FUNCTION_BLOCK CoEResetTask IMPLEMENTS I_Task, I_Cyclic, I_Object, I_Abortable, I_Abortable, I_Resettable
VAR
	mcReset : Tc2_MC2.MC_Reset;
	_Axis : REFERENCE TO Tc2_MC2.AXIS_REF;
END_VAR

{analysis -2}

METHOD Abort : HRESULT
mcReset.Execute := FALSE;
END_METHOD

PROPERTY AxisRef : reference to Axis_Ref
GET // PUBLIC
AxisRef REF= _Axis;
END_GET
SET
_Axis REF= AxisRef;
END_SET
END_PROPERTY

PROPERTY Busy : BOOL
GET
Busy := mcReset.Busy;
END_GET
END_PROPERTY

METHOD Cycle : HRESULT
VAR_INPUT
END_VAR
mcReset(Axis := _Axis);
mcReset.Execute := FALSE;
END_METHOD

PROPERTY Done : BOOL
GET
Done := mcReset.Done;
END_GET
END_PROPERTY

PROPERTY Error : BOOL
GET
Error := mcReset.Error;
END_GET
END_PROPERTY

METHOD RegisterWithParent
VAR_INPUT
	Parent	: I_HostObjects;
END_VAR
Parent.RegisterAbortable(THIS^);
Parent.RegisterCyclic(THIS^);
Parent.RegisterTask(THIS^);
Parent.RegisterResettable(THIS^);
END_METHOD

METHOD Reset : HRESULT
VAR_INPUT
END_VAR
IF mcReset.Execute THEN
	Reset := -1;
ELSE
	mcReset.Execute := TRUE;
END_IF
END_METHOD

END_FUNCTION_BLOCK

(* stored: Version 1.1.0.1
   POU CoEResetTask: Id {ea00788b-a7e2-4ddb-a987-8527d11bfcf5}, SpecialFunc None
   Method Abort: Id {175585a1-cdb8-4dd4-9630-03b10e9f2656}
   Property AxisRef: Id {b3b662e8-3ce3-48c8-a8d0-fc2d4bd302cd}
   Get Get: Id {23224859-c01c-495b-a166-81f774c86dc0}
   Set Set: Id {378228be-d0bf-44b9-a6ef-d5a5e53194bf}
   Property Busy: Id {6fd13692-80ad-4e8c-b6fa-bf24745db6e9}
   Get Get: Id {3f3da426-01ff-4963-9c05-3e4c10dc1883}
   Method Cycle: Id {a2f61a2f-8d99-4872-967a-55fbf379e9cf}
   Property Done: Id {b2c4b57c-337f-40bd-8e81-565ad6a269f2}
   Get Get: Id {214b1997-2421-46e9-bb64-09da6c6af054}
   Property Error: Id {7069ca0e-f0b0-4125-b7fe-724659e58141}
   Get Get: Id {f87457df-05b1-4857-aa40-6a1ab55ff05c}
   Method RegisterWithParent: Id {ac903c7a-36cd-4508-9b6b-75b99dd2293c}
   Method Reset: Id {3351ec6f-5e58-4cce-afac-76b6f35f5e04} *)
